_CFC_ (* Continuous Function Chart, elements in execution order *)
#0 SR_SHU6_PV1_TSMP1_DI4:SR(SET1: #1.Q, RESET: SHU6_PV1_SB)
#1 TOF_TSMP1:TOF(IN: #2, PT: t#10s)
#2 AND(NOT SHU6_PV1_Z_NET_VH_NAPR, #4.Q)
#3 SHU6_PV1_Z_MP1_TH <= #0.Q1
#4 TON1:TON(IN: NOT SHU6_PV1_TSMP1_DI4, PT: t#3s)
_END_CFC_
(* the same logic as Structured Text *)
SR_SHU6_PV1_TSMP1_DI4(SET1 := TOF_TSMP1.Q, RESET := SHU6_PV1_SB);
TOF_TSMP1(IN := _t23, PT := t#10s);
_t23 := NOT SHU6_PV1_Z_NET_VH_NAPR AND TON1.Q;
SHU6_PV1_Z_MP1_TH := SR_SHU6_PV1_TSMP1_DI4.Q1;
TON1(IN := NOT SHU6_PV1_TSMP1_DI4, PT := t#3s);
END_PROGRAM

(* POU TZBiS/TZB/Z_MV1_Avar, CFC *)
PROGRAM Z_MV1_Avar
VAR

	SR_MV1_Avar: SR;
	SR_MV2_Avar: SR;
END_VAR
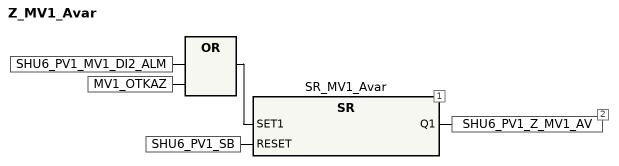
_CFC_ (* Continuous Function Chart, elements in execution order *)
#0 OR(SHU6_PV1_MV1_DI2_ALM, MV1_OTKAZ)
#1 SR_MV1_Avar:SR(SET1: #0, RESET: SHU6_PV1_SB)
#2 SHU6_PV1_Z_MV1_AV <= #1.Q1
_END_CFC_
(* the same logic as Structured Text *)
SR_MV1_Avar(SET1 := SHU6_PV1_MV1_DI2_ALM OR MV1_OTKAZ, RESET := SHU6_PV1_SB);
SHU6_PV1_Z_MV1_AV := SR_MV1_Avar.Q1;
END_PROGRAM

(* POU TZBiS/TZB/Z_MV1_NP, CFC *)
PROGRAM Z_MV1_NP
VAR
	SR_MV1_NPit: SR;
	SR_MV2_NPit: SR;
END_VAR
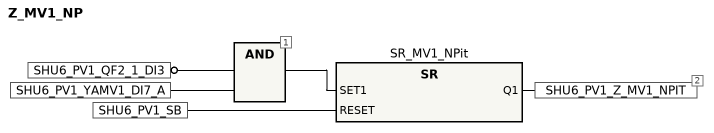
_CFC_ (* Continuous Function Chart, elements in execution order *)
#0 SR_MV1_NPit:SR(SET1: #1, RESET: SHU6_PV1_SB)
#1 AND(NOT SHU6_PV1_QF2_1_DI3, SHU6_PV1_YAMV1_DI7_A)
#2 SHU6_PV1_Z_MV1_NPIT <= #0.Q1
_END_CFC_
END_PROGRAM

(* POU TZBiS/TZB/Z_MV1_Pereg, CFC *)
PROGRAM Z_MV1_Pereg
VAR
	TON1: TON;
	TOF_TSMV1: TOF;
	SR_SHU6_PV1_TSMV1_6_1_DI6:SR;
END_VAR
VAR (* helpers for the ST form of the networks *)
	_t23 : BOOL;
END_VAR
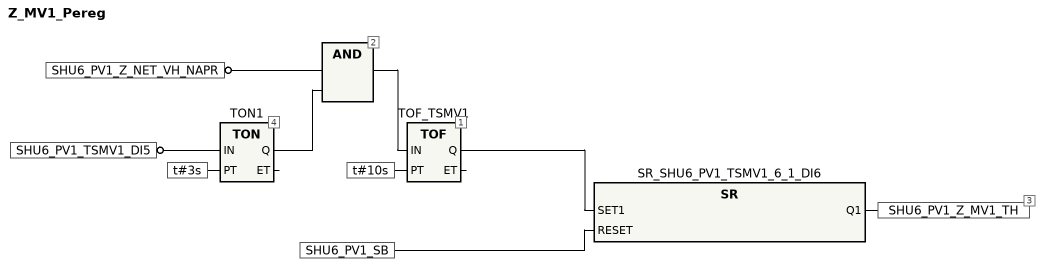
_CFC_ (* Continuous Function Chart, elements in execution order *)
#0 SR_SHU6_PV1_TSMV1_6_1_DI6:SR(SET1: #1.Q, RESET: SHU6_PV1_SB)
#1 TOF_TSMV1:TOF(IN: #2, PT: t#10s)
#2 AND(NOT SHU6_PV1_Z_NET_VH_NAPR, #4.Q)
#3 SHU6_PV1_Z_MV1_TH <= #0.Q1
#4 TON1:TON(IN: NOT SHU6_PV1_TSMV1_DI5, PT: t#3s)
_END_CFC_
(* the same logic as Structured Text *)
SR_SHU6_PV1_TSMV1_6_1_DI6(SET1 := TOF_TSMV1.Q, RESET := SHU6_PV1_SB);
TOF_TSMV1(IN := _t23, PT := t#10s);
_t23 := NOT SHU6_PV1_Z_NET_VH_NAPR AND TON1.Q;
SHU6_PV1_Z_MV1_TH := SR_SHU6_PV1_TSMV1_6_1_DI6.Q1;
TON1(IN := NOT SHU6_PV1_TSMV1_DI5, PT := t#3s);
END_PROGRAM

(* POU TZBiS/TZB/Z_MRQ1_Avar, CFC *)
PROGRAM Z_MRQ1_Avar
VAR
	SR_MRQ1_Avar: SR;
END_VAR
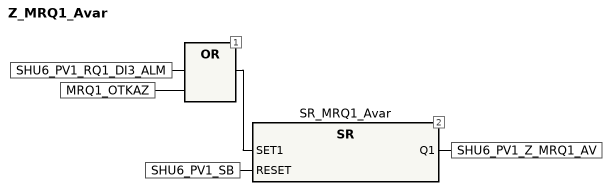
_CFC_ (* Continuous Function Chart, elements in execution order *)
#0 SHU6_PV1_Z_MRQ1_AV <= #2.Q1
#1 OR(SHU6_PV1_RQ1_DI3_ALM, MRQ1_OTKAZ)
#2 SR_MRQ1_Avar:SR(SET1: #1, RESET: SHU6_PV1_SB)
_END_CFC_
(* the same logic as Structured Text *)
SHU6_PV1_Z_MRQ1_AV := SR_MRQ1_Avar.Q1;
SR_MRQ1_Avar(SET1 := SHU6_PV1_RQ1_DI3_ALM OR MRQ1_OTKAZ, RESET := SHU6_PV1_SB);
END_PROGRAM

(* POU TZBiS/TZB/Z_MRQ1_NP, CFC *)
PROGRAM Z_MRQ1_NP
VAR
	SR_M3_NPit: SR;
END_VAR
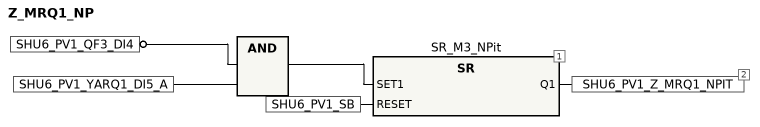
_CFC_ (* Continuous Function Chart, elements in execution order *)
#0 AND(NOT SHU6_PV1_QF3_DI4, SHU6_PV1_YARQ1_DI5_A)
#1 SR_M3_NPit:SR(SET1: #0, RESET: SHU6_PV1_SB)
#2 SHU6_PV1_Z_MRQ1_NPIT <= #1.Q1
_END_CFC_
(* the same logic as Structured Text *)
SR_M3_NPit(SET1 := NOT SHU6_PV1_QF3_DI4 AND SHU6_PV1_YARQ1_DI5_A, RESET := SHU6_PV1_SB);
SHU6_PV1_Z_MRQ1_NPIT := SR_M3_NPit.Q1;
END_PROGRAM

(* POU TZBiS/TZB/Z_NET_VKH_NAPR, CFC *)
PROGRAM Z_NET_VKH_NAPR
VAR
	RS_Net_vhk_napr: SR;
	TON_KV: TON;
END_VAR
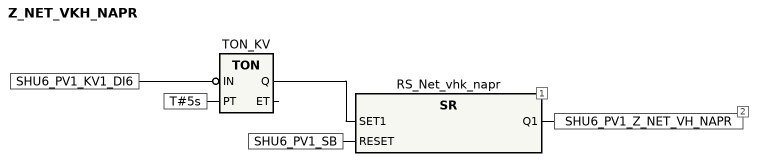
_CFC_ (* Continuous Function Chart, elements in execution order *)
#0 TON_KV:TON(IN: NOT SHU6_PV1_KV1_DI6, PT: T#5s)
#1 RS_Net_vhk_napr:SR(SET1: #0.Q, RESET: SHU6_PV1_SB)
#2 SHU6_PV1_Z_NET_VH_NAPR <= #1.Q1
_END_CFC_
(* the same logic as Structured Text *)
TON_KV(IN := NOT SHU6_PV1_KV1_DI6, PT := T#5s);
RS_Net_vhk_napr(SET1 := TON_KV.Q, RESET := SHU6_PV1_SB);
SHU6_PV1_Z_NET_VH_NAPR := RS_Net_vhk_napr.Q1;
END_PROGRAM

(* POU TZBiS/TZB/Z_NP_MP1, CFC *)
PROGRAM Z_NP_MP1
VAR
	TON_PDS2: TON;
	TON_ReRab: TON;
	TON_MVKL: TON;
	TON_AVT: TON;
	TP_SR: TP;
	SR_NP_M1: SR;
	SR_NP_M2: SR;
	TON_MVKL_M1: TON;
	TON_AVT_M1: TON;
	TON_AVT_M2: TON;
	TON_MVKL_M2: TON;
END_VAR
VAR (* helpers for the ST form of the networks *)
	_t70 : BOOL;
END_VAR
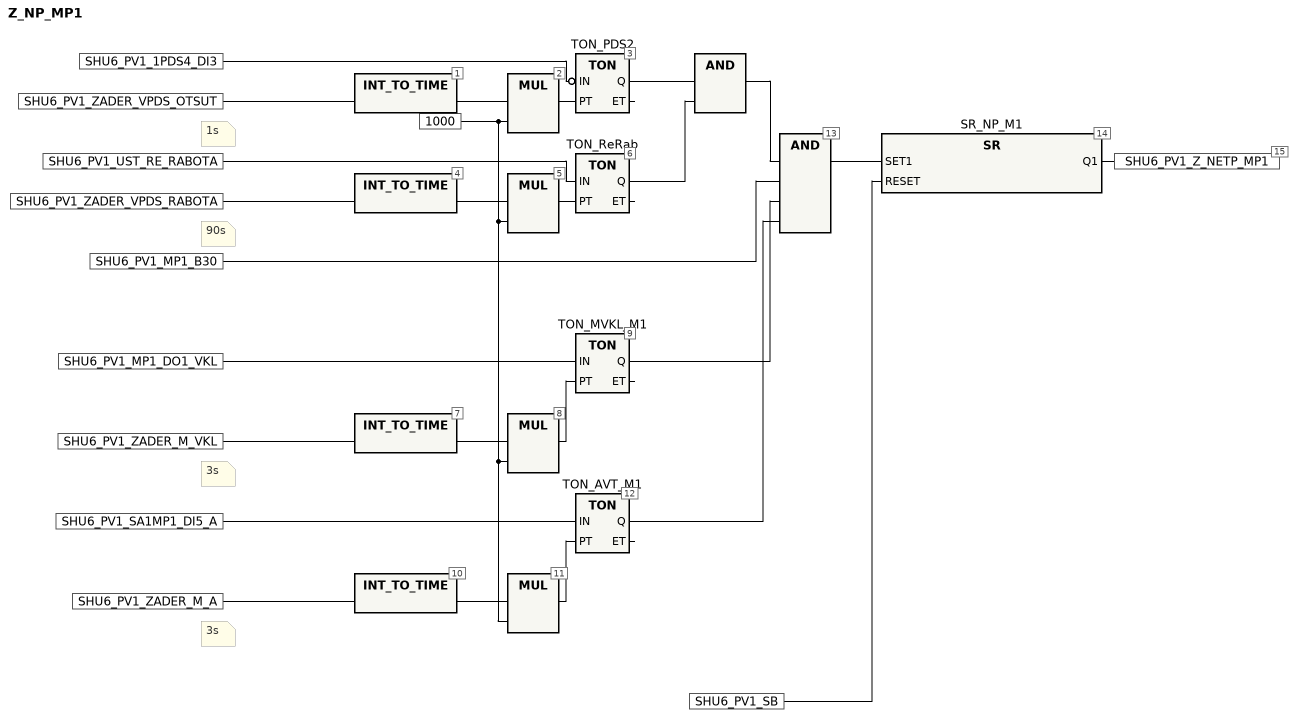
_CFC_ (* Continuous Function Chart, elements in execution order *)
(* 3s *)
(* 3s *)
(* 90s *)
(* 1s *)
#0 AND(#3.Q, #6.Q)
#1 INT_TO_TIME(SHU6_PV1_ZADER_VPDS_OTSUT)
#2 MUL(#1, 1000)
#3 TON_PDS2:TON(IN: NOT SHU6_PV1_1PDS4_DI3, PT: #2)
#4 INT_TO_TIME(SHU6_PV1_ZADER_VPDS_RABOTA)
#5 MUL(#4, 1000)
#6 TON_ReRab:TON(IN: SHU6_PV1_UST_RE_RABOTA, PT: #5)
#7 INT_TO_TIME(SHU6_PV1_ZADER_M_VKL)
#8 MUL(#7, 1000)
#9 TON_MVKL_M1:TON(IN: SHU6_PV1_MP1_DO1_VKL, PT: #8)
#10 INT_TO_TIME(SHU6_PV1_ZADER_M_A)
#11 MUL(#10, 1000)
#12 TON_AVT_M1:TON(IN: SHU6_PV1_SA1MP1_DI5_A, PT: #11)
#13 AND(#0, SHU6_PV1_MP1_B30, #9.Q, #12.Q)
#14 SR_NP_M1:SR(SET1: #13, RESET: SHU6_PV1_SB)
#15 SHU6_PV1_Z_NETP_MP1 <= #14.Q1
_END_CFC_
(* the same logic as Structured Text *)
(* 3s *)
(* 3s *)
(* 90s *)
(* 1s *)
_t70 := TON_PDS2.Q AND TON_ReRab.Q;
TON_PDS2(IN := NOT SHU6_PV1_1PDS4_DI3, PT := INT_TO_TIME(SHU6_PV1_ZADER_VPDS_OTSUT) * 1000);
TON_ReRab(IN := SHU6_PV1_UST_RE_RABOTA, PT := INT_TO_TIME(SHU6_PV1_ZADER_VPDS_RABOTA) * 1000);
TON_MVKL_M1(IN := SHU6_PV1_MP1_DO1_VKL, PT := INT_TO_TIME(SHU6_PV1_ZADER_M_VKL) * 1000);
TON_AVT_M1(IN := SHU6_PV1_SA1MP1_DI5_A, PT := INT_TO_TIME(SHU6_PV1_ZADER_M_A) * 1000);
SR_NP_M1(SET1 := _t70 AND SHU6_PV1_MP1_B30 AND TON_MVKL_M1.Q AND TON_AVT_M1.Q, RESET := SHU6_PV1_SB);
SHU6_PV1_Z_NETP_MP1 := SR_NP_M1.Q1;
END_PROGRAM

(* POU TZBiS/TZB/Z_NP_MV1, CFC *)
PROGRAM Z_NP_MV1
VAR
	TON_PDS2: TON;
	TON_ReRab: TON;
	TON_MVKL: TON;
	TON_AVT: TON;
	TP_SR: TP;
	SR_NP_M1: SR;
	SR_NP_M2: SR;
	TON_MVKL_M1: TON;
	TON_AVT_M1: TON;
	TON_AVT_M2: TON;
	TON_MVKL_M2: TON;
	SR_NP_MV1: SR;
	SR_NP_MV2: SR;
	TON_PDS3: TON;
	TON_MVKL_MV1: TON;
	TON_AVT_MV1: TON;
	TON_MVKL_MV2: TON;
	TON_AVT_MV2: TON;
END_VAR
VAR (* helpers for the ST form of the networks *)
	_t70 : BOOL;
END_VAR
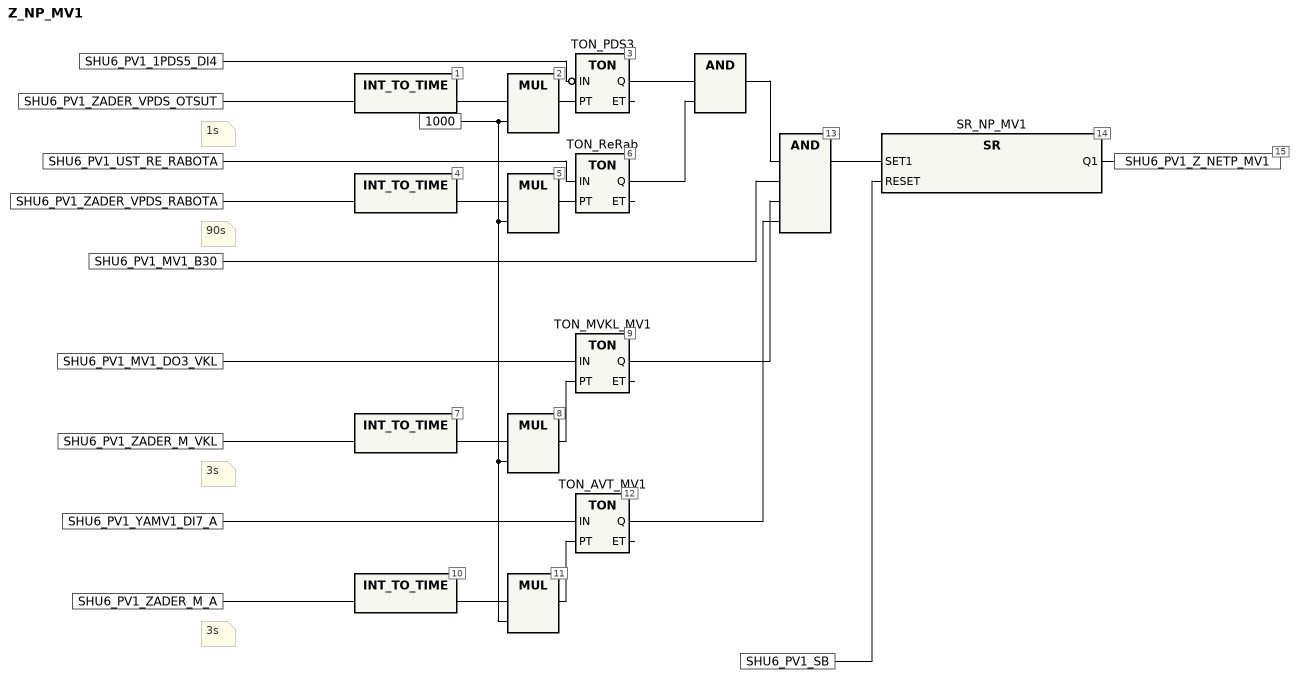
